ABB RobotStudio station: project_template.rspag

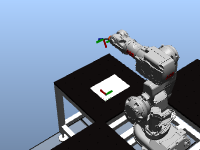
--- station ---
Station project_template (saved by RobotStudio 7.0.8504.151)
Controller IRB_140_6kg_0.81m, task T_ROB1: task frame (RAPID world) sits at (0, 0, 670) mm in the station
Controller IRB_140_6kg_0.81m
  mechanical unit ROB_1: IRB140_6_81_C_03, 6 joints, base frame (0, 0, 0) mm
Layout (positions relative to the parent item):
  - IRB140_6_81_C_03 [mechanism, from Robots\IRB140_6_81_C_G_03.rslib] at (0, 0, 670) mm; joint values [0, 0, 0, 0, 0.5236, 0] (rad or m)
  - paper [part, from Lab1 Pen\paper.rslib]
  - pen [mechanism, from Lab1 Pen\pen.rslib] at (506.29, 0, 1349.5) mm, rotated rx 180 ry 60 rz 180 deg
  - rob-table [part, from Lab1 Pen\rob-table.rslib]
Attachment: pen is attached to IRB140_6_81_C_03 / Link6
Targets, tools, work objects and paths stored in the station and not in the controller backup, written as RAPID:
! task T_ROB1
MODULE CalibData
  PERS tooldata pen:=[TRUE,[[0,0,139],[1,0,0,0]],[0.5,[0,0,20],[1,0,0,0],0,0,0]];
  TASK PERS wobjdata Workobject_1:=[FALSE,TRUE,"",[[450,125,116],[0,1,0,0]],[[50,50,-15],[1,0,0,0]]];
ENDMODULE


--- Backups/IRB_140_6kg_0.81m/RAPID/TASK1/PROGMOD/Module1.mod ---
MODULE Module1
    !***********************************************************
    !
    ! Module:  Module1
    !
    ! Description:
    !   <Insert description here>
    !
    ! Author: jo6402en-s
    !
    ! Version: 1.0
    !
    !***********************************************************


    !***********************************************************
    !
    ! Procedure main
    !
    !   This is the entry point of your program
    !
    !***********************************************************
    PROC main()
        !Add your code here
    ENDPROC
ENDMODULE
